{attribute 'GeneratedUsingTerminal: EK1122-0000-0018'}
{attribute addProperty BoxType "EK1122-0000-0018"}
{attribute addProperty Id "Beckhoff_EL32xxsub_EK1100EK1100_AB5A94672"}
{attribute addProperty CRC "1757639791"}
{attribute addProperty Size "2"}
TYPE Beckhoff_EL32xxEK1122_68C3746F EXTENDS EK1122_AB5A9467 :
STRUCT
	{attribute addProperty Name "Beckhoff_EL32xxsub_EK1100"}
	Beckhoff_EL32xxsub_EK1100 : EK1100_AB5A9467;
END_STRUCT
END_TYPE

(* stored: Version 1.2.0.0, ProductVersion 3.1.4024.9
   DUT Beckhoff_EL32xxEK1122_68C3746F: Id {c2bb5ed7-df24-4f45-8d90-7ed905fd7954} *)
